FUNCTION SaveInMemory : BOOL
VAR_INPUT
    sData : REFERENCE TO STRING(2000);
END_VAR
VAR
    fbJson     : FB_JsonSaxWriter;
    i          : int;
END_VAR

fbJson.ResetDocument();

// array1
fbJson.StartObject();
fbJson.AddKey('StationTime1');
fbJson.StartArray();

FOR i := 1 TO CONST.STATION_NUMBER BY 1 DO
    fbJson.AddDint(PERS.iStationTimeDef1[i]);
END_FOR

fbJson.EndArray();
fbJson.EndObject();

// array2
fbJson.StartObject();
fbJson.AddKey('StationTime2');
fbJson.StartArray();

FOR i := 1 TO CONST.STATION_NUMBER BY 1 DO
    fbJson.AddDint(PERS.iStationTimeDef2[i]);
END_FOR

fbJson.EndArray();
fbJson.EndObject();

// end of file
sData := fbJson.GetDocument();

fbJson.ResetDocument();

END_FUNCTION

(* stored: Version 1.1.0.1, ProductVersion 3.1.4024.6
   POU SaveInMemory: Id {775105ca-9365-4054-8101-5ff720f6736e}, SpecialFunc None *)
